PROGRAM MAPPING_out
VAR CONSTANT
{IF defined (AXIS_MAP)}
  {info 'MAPPING_out - ACTIVE'}
  bBypassMapping    : BOOL  := FALSE;
{ELSE}
  bBypassMapping    : BOOL  := TRUE;
{END_IF}
END_VAR
VAR
{IF defined (AXIS_MAP)}
  AxisState         : U_AXIS_STATE;
  AxisInfo          : U_AXIS_INFO;
  AxisParameterRd   : U_AXIS_NC_PARAMETER_RD;
{ELSE}
  AxisState         : BYTE;
  AxisInfo          : BYTE;
  AxisParameterRd   : BYTE;
{END_IF}
END_VAR

IF bBypassMapping THEN RETURN; END_IF

memcpy(ADR(AxisState),         ADR(GVL_AXIS.State),             SIZEOF(GVL_AXIS.State));
memcpy(ADR(AxisInfo),          ADR(GVL_AXIS.Info),              SIZEOF(GVL_AXIS.Info));
memcpy(ADR(AxisParameterRd),   ADR(GVL_AXIS.NcParameterRd),     SIZEOF(GVL_AXIS.NcParameterRd));

END_PROGRAM

(* stored: Version 1.1.0.1, ProductVersion 3.1.4024.12
   POU MAPPING_out: Id {f452c8f5-5dcb-0f99-160c-afb3c9dfaf6c}, SpecialFunc None *)
